VAR_GLOBAL

	ProximitySensorX			AT%I*		:	BOOL;
	ProximitySensorY			AT%I*		:	BOOL;
	ProximitySensorZ			AT%I*		:	BOOL;



END_VAR

(* stored: Version 1.1.0.1
   GVL IO: Id {5c633ecf-caed-058c-1a16-2b1fdf36f8a0} *)
